TYPE "ITF_A01"
VERSION : 0.1
// Block: ITF_A01
   STRUCT
      aa : Bool;
   END_STRUCT;

END_TYPE

